(*
    In this testsuite we are running the same testcase over two cycles, and thus calling every assert method twice.
    This is in order to verify that we don't print every FAILED assert twice.
*)
{attribute 'call_after_init'}
FUNCTION_BLOCK FB_AssertEveryFailedTestTwice EXTENDS TcUnit.FB_TestSuite IMPLEMENTS TcUnit.I_RunnableTestSuite
VAR
    Assert : TcUnit.FB_Assert;
    AssertCount : USINT := 0;
END_VAR

METHOD FB_init : BOOL
VAR_INPUT
	bInitRetains : BOOL; // if TRUE, the retain variables are initialized (warm start / cold start)
	bInCopyCode : BOOL;  // if TRUE, the instance afterwards gets moved into the copy code (online change)
END_VAR
SUPER^.RegisterTestSuite(THIS^);
END_METHOD

METHOD RunTests : TCUNIT.E_TestSuiteRunState
TwiceAssertCall();

AssertCount := AssertCount + 1;
IF AssertCount = 2 THEN
    RunTests := TCUNIT.E_TestSuiteRunState.FINISHED;
END_IF
END_METHOD

METHOD PRIVATE TwiceAssertCall
VAR
    aANY : INT := 55;
    bANY : INT := 77;

    aBOOL : BOOL := TRUE;
    bBOOL : BOOL := FALSE;

    aBYTE : BYTE := 16#AB;
    bBYTE : BYTE := 16#BA;

    aDATE : DATE := DATE#1996-05-06;
    bDATE : DATE := DATE#2019-01-20;

    aDATE_AND_TIME : DATE_AND_TIME := DATE_AND_TIME#1996-05-06-15:36:30;
    bDATE_AND_TIME : DATE_AND_TIME := DATE_AND_TIME#1972-03-29-00:00:00;

    aDINT : DINT := 4444;
    bDINT : DINT := 3333;

    aDWORD : DWORD := 16#AAAAAAAA;
    bDWORD : DWORD := 16#BBBBBBBB;

    aINT : INT := 30000;
    bINT : INT := 32000;

    aLINT : LINT := 50000;
    bLINT : LINT := 50001;

    aLREAL : LREAL := 33.3;
    bLREAL : LREAL := 44.4;

    aLTIME : LTIME := LTIME#213503D23H34M33S709MS551US615NS;
    bLTIME : LTIME := LTIME#1000D15H23M12S34MS2US44NS;

    aLWORD : LWORD := 16#AAAAAAAAAAAAAAAA;
    bLWORD : LWORD := 16#BBBBBBBBBBBBBBBB;

    aREAL : REAL := 44.4;
    bREAL : REAL := 22.2;

    aSINT : SINT := 99;
    bSINT : SINT := 10;

    aSTRING : STRING := 'Hello world';
    bSTRING : STRING := 'Hey there';

    aUDINT : UDINT := 249494994;
    bUDINT : UDINT := 1223;

    aUINT : UINT := 3444;
    bUINT : UINT := 3445;

    aULINT : ULINT := 789234475;
    bULINT : ULINT := 34523327234;

    aUSINT : USINT := 34;
    bUSINT : USINT := 36;

    aTIME : TIME := T#12H34M15S10MS;
    bTIME : TIME := T#11H34M13S244MS;

    aTIME_OF_DAY : TIME_OF_DAY := TIME_OF_DAY#15:36:30.123;
    bTIME_OF_DAY : TIME_OF_DAY := TIME_OF_DAY#06:21:11.492;

    aWORD : WORD := 16#ABCD;
    bWORD : WORD := 16#89EF;
END_VAR
TEST('TwiceAssertCall');

Assert.AssertEquals(Expected := aANY,
                    Actual := bANY,
                    Message := 'Not equal ANY');
                    
Assert.AssertEquals_BOOL(Expected := aBOOL,
                         Actual := bBOOL,
                         Message := 'Not equal BOOL');

Assert.AssertEquals_BYTE(Expected := aBYTE,
                         Actual := bBYTE,
                         Message := 'Not equal BYTE');

Assert.AssertEquals_DATE(Expected := aDATE,
                         Actual := bDATE,
                         Message := 'Not equal DATE');

Assert.AssertEquals_DATE_AND_TIME(Expected := aDATE_AND_TIME,
                                  Actual := bDATE_AND_TIME,
                                  Message := 'Not equal DATE_AND_TIME');

Assert.AssertEquals_DINT(Expected := aDINT,
                         Actual := bDINT,
                         Message := 'Not equal DINT');

Assert.AssertEquals_DWORD(Expected := aDWORD,
                          Actual := bDWORD,
                          Message := 'Not equal DWORD');

Assert.AssertEquals_INT(Expected := aINT,
                        Actual := bINT,
                        Message := 'Not equal INT');

Assert.AssertEquals_LINT(Expected := aLINT,
                         Actual := bLINT,
                         Message := 'Not equal LINT');

Assert.AssertEquals_LREAL(Expected := aLREAL,
                         Actual := bLREAL,
                         Delta := 0.1,
                         Message := 'Not equal LREAL');

Assert.AssertEquals_LTIME(Expected := aLTIME,
                          Actual := bLTIME,
                          Message := 'Not equal LTIME');

Assert.AssertEquals_LWORD(Expected := aLWORD,
                          Actual := bLWORD,
                          Message := 'Not equal LWORD');

Assert.AssertEquals_REAL(Expected := aREAL,
                          Actual := bREAL,
                          Delta := 0.1,
                          Message := 'Not equal REAL');

Assert.AssertEquals_SINT(Expected := aSINT,
                          Actual := bSINT,
                          Message := 'Not equal SINT');

Assert.AssertEquals_STRING(Expected := aSTRING,
                           Actual := bSTRING,
                           Message := 'Not equal STRING');

Assert.AssertEquals_UDINT(Expected := aUDINT,
                           Actual := bUDINT,
                           Message := 'Not equal UDINT');

Assert.AssertEquals_UINT(Expected := aUINT,
                         Actual := bUINT,
                         Message := 'Not equal UINT');

Assert.AssertEquals_ULINT(Expected := aULINT,
                          Actual := bULINT,
                          Message := 'Not equal ULINT');

Assert.AssertEquals_USINT(Expected := aUSINT,
                          Actual := bUSINT,
                          Message := 'Not equal USINT');

Assert.AssertEquals_TIME(Expected := aTIME,
                         Actual := bTIME,
                         Message := 'Not equal TIME');

Assert.AssertEquals_TIME_OF_DAY(Expected := aTIME_OF_DAY,
                                Actual := bTIME_OF_DAY,
                                Message := 'Not equal TIME_OF_DAY');

Assert.AssertEquals_WORD(Expected := aWORD,
                          Actual := bWORD,
                          Message := 'Not equal WORD');
END_METHOD

END_FUNCTION_BLOCK

(* stored: Version 1.1.0.1, ProductVersion 3.1.4022.16
   POU FB_AssertEveryFailedTestTwice: Id {3bea6e4d-8d08-467b-90da-24a784807eae}, SpecialFunc None
   Method FB_init: Id {ec220df4-f39f-4ff5-8348-a9f7930e9f4a}
   Method RunTests: Id {67907b15-cc1a-4b64-8465-b6b1fd17bd6d}
   Method TwiceAssertCall: Id {69d3987a-7ce5-4206-ac7a-879b67c9a54d} *)
